(* CODESYS project Group11_Ass2.export

Project tree, tasks and I/O mapping:
  control/
    function block DoorCtrl [SFC]
    program ElevatorControl [LD]
    program main [ST]
*)

// control/DoorCtrl
FUNCTION_BLOCK DoorCtrl
VAR_INPUT
	open: BOOL;
	precondition: BOOL;
	forceClose: BOOL;
	openedSensor: BOOL;
	closedSensor: BOOL;
	
	OpenAutomatically: BOOL;
	RequestElevator: BOOL;
END_VAR
VAR_OUTPUT
	executing: BOOL;
	closed: BOOL;
	openControl: BOOL;
END_VAR
VAR
END_VAR

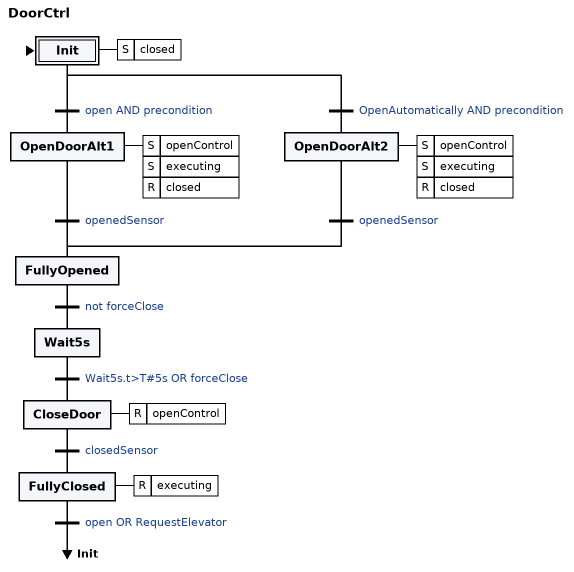
INITIAL_STEP Init:
    closed(S);
END_STEP
TRANSITION FROM Init TO OpenDoorAlt1
    := open AND precondition;
END_TRANSITION
STEP OpenDoorAlt1:
    openControl(S);
    executing(S);
    closed(R);
END_STEP
TRANSITION FROM OpenDoorAlt1 TO FullyOpened
    := openedSensor;
END_TRANSITION
TRANSITION FROM Init TO OpenDoorAlt2
    := OpenAutomatically AND precondition;
END_TRANSITION
STEP OpenDoorAlt2:
    openControl(S);
    executing(S);
    closed(R);
END_STEP
TRANSITION FROM OpenDoorAlt2 TO FullyOpened
    := openedSensor;
END_TRANSITION
STEP FullyOpened:
END_STEP
TRANSITION FROM FullyOpened TO Wait5s
    := not forceClose;
END_TRANSITION
STEP Wait5s:
END_STEP
TRANSITION FROM Wait5s TO CloseDoor
    := Wait5s.t>T#5s OR forceClose;
END_TRANSITION
STEP CloseDoor:
    openControl(R);
END_STEP
TRANSITION FROM CloseDoor TO FullyClosed
    := closedSensor;
END_TRANSITION
STEP FullyClosed:
    executing(R);
END_STEP
TRANSITION FROM FullyClosed TO Init
    := open OR RequestElevator;
END_TRANSITION

END_FUNCTION_BLOCK

// control/ElevatorControl
PROGRAM ElevatorControl
VAR
	up: BOOL;
	down: BOOL;

	requestF1: BOOL;
	requestF2: BOOL;
	requestF3: BOOL;
	requestF4: BOOL := TRUE;

	GoDown: BOOL;
	GoUp: BOOL := TRUE;
	
	DoorsF4: DoorCtrl;
	DoorsF3: DoorCtrl;
	DoorsF2: DoorCtrl;
	DoorsF1: DoorCtrl;
	
	DoorIsClosed: BOOL;
	AutoOpen: BOOL;
	ElevatorRequested: BOOL;
	
	GoingUp: BOOL;
	GoingDown: BOOL;
END_VAR
VAR // added by the converter: edge detectors and wires of the graphical bodies
    _w1, _w2, _w3, _w4, _w5, _w6 : BOOL;
    _ft1, _ft2, _ft3, _ft4 : F_TRIG;
END_VAR

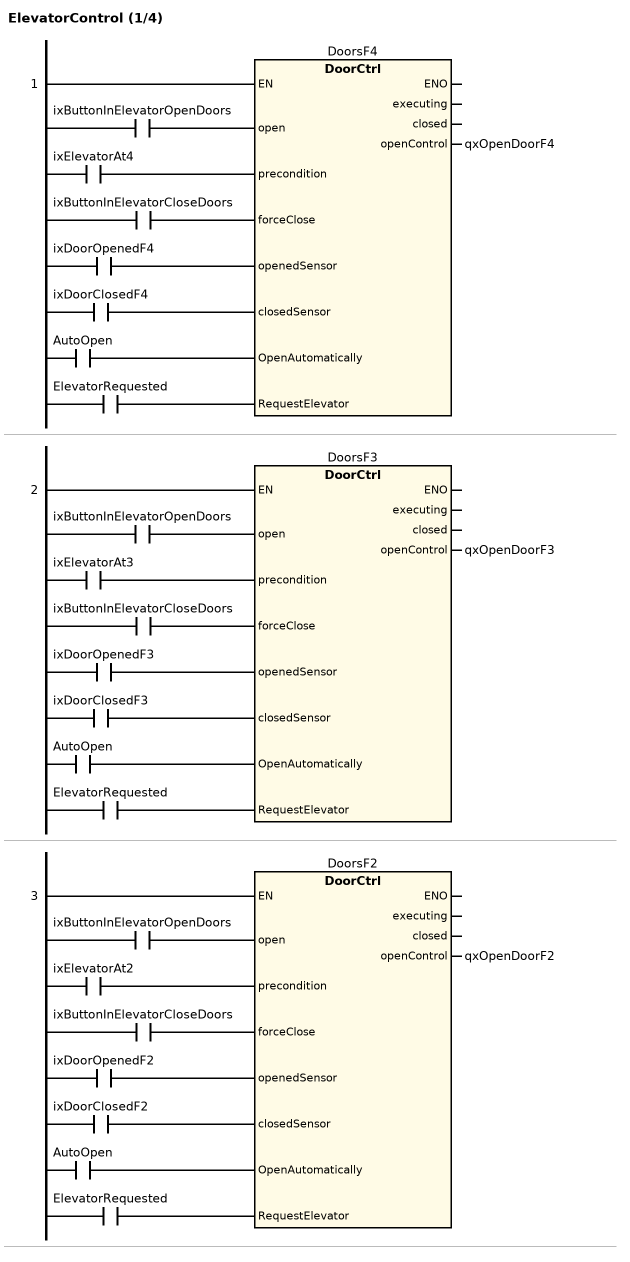
// NETWORK 1
DoorsF4(
    open := ixButtonInElevatorOpenDoors,
    precondition := ixElevatorAt4,
    forceClose := ixButtonInElevatorCloseDoors,
    openedSensor := ixDoorOpenedF4,
    closedSensor := ixDoorClosedF4,
    OpenAutomatically := AutoOpen,
    RequestElevator := ElevatorRequested,
    openControl => qxOpenDoorF4); // DoorCtrl

// NETWORK 2
DoorsF3(
    open := ixButtonInElevatorOpenDoors,
    precondition := ixElevatorAt3,
    forceClose := ixButtonInElevatorCloseDoors,
    openedSensor := ixDoorOpenedF3,
    closedSensor := ixDoorClosedF3,
    OpenAutomatically := AutoOpen,
    RequestElevator := ElevatorRequested,
    openControl => qxOpenDoorF3); // DoorCtrl

// NETWORK 3
DoorsF2(
    open := ixButtonInElevatorOpenDoors,
    precondition := ixElevatorAt2,
    forceClose := ixButtonInElevatorCloseDoors,
    openedSensor := ixDoorOpenedF2,
    closedSensor := ixDoorClosedF2,
    OpenAutomatically := AutoOpen,
    RequestElevator := ElevatorRequested,
    openControl => qxOpenDoorF2); // DoorCtrl

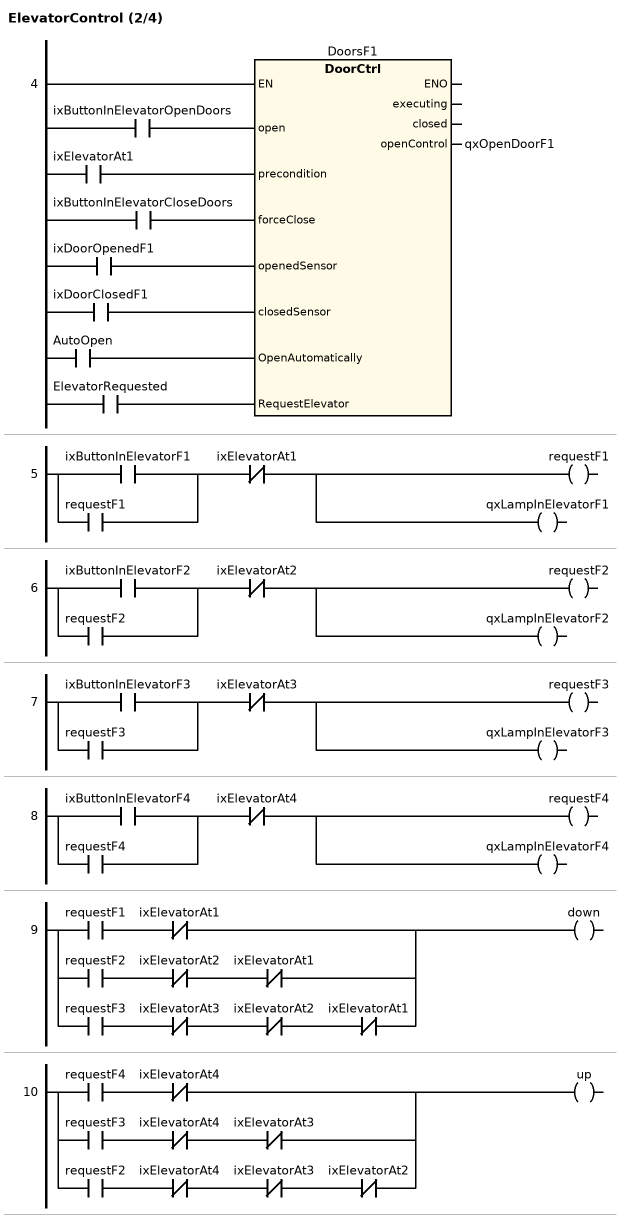
// NETWORK 4
DoorsF1(
    open := ixButtonInElevatorOpenDoors,
    precondition := ixElevatorAt1,
    forceClose := ixButtonInElevatorCloseDoors,
    openedSensor := ixDoorOpenedF1,
    closedSensor := ixDoorClosedF1,
    OpenAutomatically := AutoOpen,
    RequestElevator := ElevatorRequested,
    openControl => qxOpenDoorF1); // DoorCtrl

// NETWORK 5
_w1 := (ixButtonInElevatorF1 OR requestF1) AND NOT ixElevatorAt1;
requestF1 := _w1;
qxLampInElevatorF1 := _w1;

// NETWORK 6
_w2 := (ixButtonInElevatorF2 OR requestF2) AND NOT ixElevatorAt2;
requestF2 := _w2;
qxLampInElevatorF2 := _w2;

// NETWORK 7
_w3 := (ixButtonInElevatorF3 OR requestF3) AND NOT ixElevatorAt3;
requestF3 := _w3;
qxLampInElevatorF3 := _w3;

// NETWORK 8
_w4 := (ixButtonInElevatorF4 OR requestF4) AND NOT ixElevatorAt4;
requestF4 := _w4;
qxLampInElevatorF4 := _w4;

// NETWORK 9
down := requestF1 AND NOT ixElevatorAt1 OR requestF2 AND NOT ixElevatorAt2 AND NOT ixElevatorAt1 OR requestF3 AND NOT ixElevatorAt3 AND NOT ixElevatorAt2 AND NOT ixElevatorAt1;

// NETWORK 10
up := requestF4 AND NOT ixElevatorAt4 OR requestF3 AND NOT ixElevatorAt4 AND NOT ixElevatorAt3 OR requestF2 AND NOT ixElevatorAt4 AND NOT ixElevatorAt3 AND NOT ixElevatorAt2;

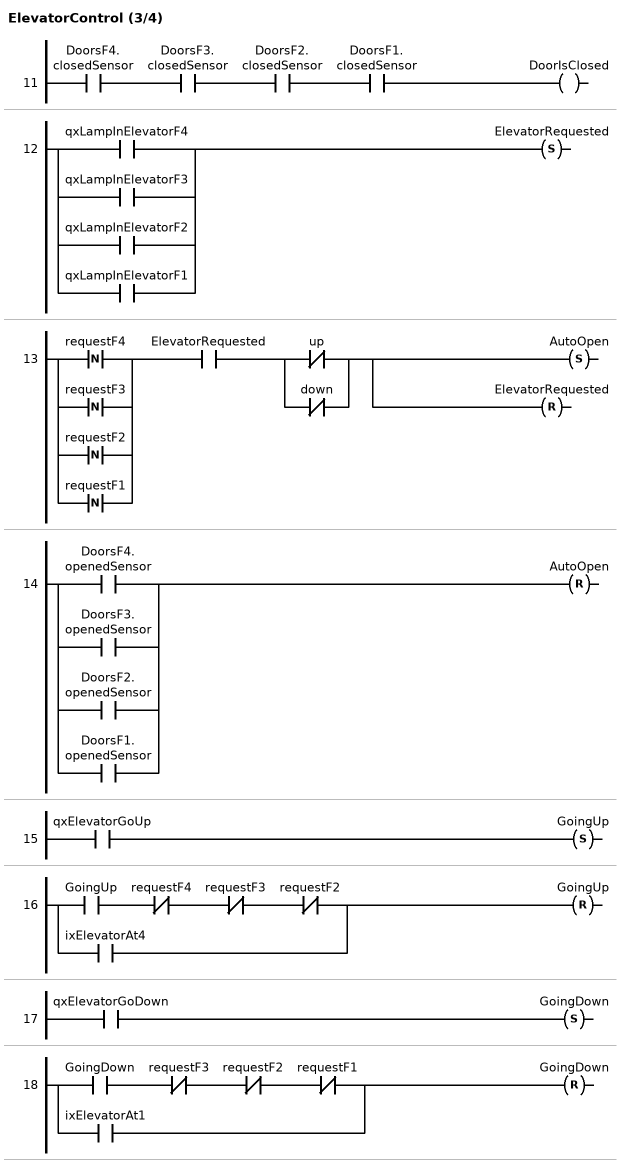
// NETWORK 11
DoorIsClosed := DoorsF4.closedSensor AND DoorsF3.closedSensor AND DoorsF2.closedSensor AND DoorsF1.closedSensor;

// NETWORK 12
ElevatorRequested S= qxLampInElevatorF4 OR qxLampInElevatorF3 OR qxLampInElevatorF2 OR qxLampInElevatorF1;

// NETWORK 13
_ft1(CLK := requestF4);
_ft2(CLK := requestF3);
_ft3(CLK := requestF2);
_ft4(CLK := requestF1);
_w5 := (_ft1.Q OR _ft2.Q OR _ft3.Q OR _ft4.Q) AND ElevatorRequested;
_w6 := _w5 AND NOT up OR _w5 AND NOT down;
AutoOpen S= _w6;
ElevatorRequested R= _w6;

// NETWORK 14
AutoOpen R= DoorsF4.openedSensor OR DoorsF3.openedSensor OR DoorsF2.openedSensor OR DoorsF1.openedSensor;

// NETWORK 15
GoingUp S= qxElevatorGoUp;

// NETWORK 16
GoingUp R= GoingUp AND NOT requestF4 AND NOT requestF3 AND NOT requestF2 OR ixElevatorAt4;

// NETWORK 17
GoingDown S= qxElevatorGoDown;

// NETWORK 18
GoingDown R= GoingDown AND NOT requestF3 AND NOT requestF2 AND NOT requestF1 OR ixElevatorAt1;

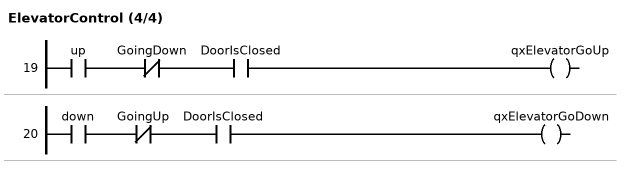
// NETWORK 19
qxElevatorGoUp := up AND NOT GoingDown AND DoorIsClosed;

// NETWORK 20
qxElevatorGoDown := down AND NOT GoingUp AND DoorIsClosed;

END_PROGRAM

// control/main
PROGRAM main
VAR
END_VAR

ElevatorControl();

END_PROGRAM
